// SIMATIC S7-200 SMART project (STEP 7-Micro/WIN SMART), CPU ST20

SYMBOL_TABLE Real_Sym
PressureDINT     VD100
PressureReal     VD104
PressRawMin      VD108
PressRawMax      VD112
PressFinalMin    VD116
PressFinalMax    VD120
PressureFinalVal VD124
TempDINT         VD128
TempReal         VD132
TempRawMin       VD136
TempRawMax       VD140
TempFinalMin     VD144
TempFinalMax     VD148
TempFinalVal     VD152
AutoPressureSV   VD156
AutoTempSV       VD160
NormPressSV      VD164
NormTempSV       VD168
RapidPressSV     VD172
RapidTempSV      VD176
OptPressSV       VD180
OptTempSV        VD184
TempErrorVal     VD188
TempErrorVal2    VD192
TempErrorValDINT VD196
HeaterOffTemp    VD200
PressureReal1    VD204
TempReal1        VD208
TempFinal1       VD212
PressureFinal1   VD216
VCCTolerance     VD220
VacuumLimit      VD224
VLTPressSV       VD228
TempRealPrint    VD232
TempDINTPrint    VD236
PressRealPrint   VD240
PressDINTPrint   VD244
END_SYMBOL_TABLE

SYMBOL_TABLE System Symbols
Always_On        SM0.0    // Always ON
Clock_1s         SM0.5    // Clock pulse that is ON for 0.5 s, OFF for 0.5 s, for a duty cycle time of 1 s.
END_SYMBOL_TABLE

SYMBOL_TABLE Bool_Sym
AutoSel          M0.0
ManualSel        M0.1
VacPumpManCmd    M0.2
HeaterManCmd     M0.3
AirVentManCmd    M0.4
PunchDownManCmd  M0.5
PunchUpManCmd    M0.6
VacPumpAutoCmd   M1.0
HeaterAutoCmd    M1.1
AirVentAutoCmd   M1.2
PunchDownAutoCmd M1.3
PunchUpAutoCmd   M1.4
AlarmCmd         M1.5
NormalSel        M2.0
RapidSel         M2.1
OptChoiceSel     M2.2
VLTSel           M2.3
AutoStart        M2.4
StartHeaterAuto  M2.5
PreTreat         M2.6
Vacuum1Done      M2.7
HeatingDone      M3.0
Vacuum2Done      M3.1
Sterilization    M3.2
Aeration         M3.3
VentOut          M3.4
CycleDone        M3.5
Vacuum3Done      M3.6
StartPunch       M3.7
PunchDone        M4.0
CycleDoneFinal   M4.1
StopOut          M4.2
OutVar           M4.3
StartHoldTime    M4.4
VLTPass          M4.5
VLTFail          M4.6
HoldTimeDone     M4.7
ResetCycleCount  M5.0
VLTStart         M5.1
VLTDone          M5.2
VLTVacuuming     M5.3
VLTHoldStart     M5.4
VLTTestPass      M5.5
VLTTestFail      M5.6
VLTDoneFinal     M5.7
MBUs_Done        M6.0
END_SYMBOL_TABLE

SYMBOL_TABLE Int_Sym
AutoSterTimeSV   VW0
AutoAerateTimeSV VW2
NormSterTimeSV   VW4
NormAerateTimeSV VW6
RapidSterTimeSV  VW8
RapidAerateTimeSV VW10
OptSterTimeSV    VW12
OptAerateTimeSV  VW14
SterTimePV       VW16
AerateTimePV     VW18
TempErrorValInt  VW20
TempBlinkOffVal  VW22
TempBlinkOffTime VW24
TempBlinkOnTime  VW26
AerateTimeSecPV  VW28
SterTimeSecPV    VW30
PunchSV          VW32
PunchPV          VW34
ClockVar1        VW36
OnCount          VW38
OffCount         VW40
VacuumHoldTimeSV VW42
VacuumHoldTimePV VW44
HoldTimePVSec    VW46
AutoStatus       VW48
CycleCount       VW50
OptHoldTimeSV    VW52
AutoHoldTimeSV   VW54
NormHoldTimeSV   VW56
RapidHoldTimeSV  VW58
TempIntPrint     VW60
PressIntPrint    VW62
YearRead         VW1774
MonthRead        VW1778
DateRead         VW1782
HourRead         VW1762
MinuteRead       VW1766
SecondsRead      VW1770
MinutesSet       VW1460
SecondsSet       VW1462
HourSet          VW1464
YearSet          VW1470
MonthSet         VW1474
DateSet          VW1490
END_SYMBOL_TABLE

ORGANIZATION_BLOCK MAIN:OB1
TITLE=Program Comments
BEGIN
Network 1
// Network Comment
LD     Always_On:SM0.0
ITD    EM0_Input0:AIW16, PressureDINT:VD100
AENO
DTR    PressureDINT:VD100, PressureReal1:VD204
AENO
MOVR   PressureReal1:VD204, PressureReal:VD104
AENO
/R     100.0, PressureReal:VD104
AENO
CALL   Lin_Trafo:SBR1, PressureReal:VD104, PressRawMin:VD108, PressRawMax:VD112, PressFinalMin:VD116, PressFinalMax:VD120, PressureFinal1:VD216
Network 2
// Network Comment
LD     Always_On:SM0.0
ITD    EM0_Input1:AIW18, TempDINT:VD128
AENO
DTR    TempDINT:VD128, TempReal1:VD208
AENO
MOVR   TempReal1:VD208, TempReal:VD132
AENO
/R     100.0, TempReal:VD132
AENO
CALL   Lin_Trafo:SBR1, TempReal:VD132, TempRawMin:VD136, TempRawMax:VD140, TempFinalMin:VD144, TempFinalMax:VD148, TempFinal1:VD212
Network 3
// (network saved uncompiled; FBD cells follow)
// row 0: c5 [INC_W ]  c8 [MOV_R ]
// row 1: c1 [AND Always_On:SM0.0 Clock_1s:SM0.5 ]  c2 --  c3 [P ]  c4 --  c5 [ EN:=power@row1, IN:=ClockVar1:VW36, ENO=>power, OUT=>ClockVar1:VW36]  c6 --  c7 --  c8 [ EN:=power@row1, IN:=TempFinal1:VD212, ENO=>V?0, OUT=>TempFinalVal:VD152]
// row 2: c1 [box]  c5 [box]  c8 [box]
Network 4
// (network saved uncompiled; FBD cells follow)
// row 0: c5 [MOV_R ]  c8 [MOV_W ]
// row 1: c1 [>=I ClockVar1:VW36 2 ]  c2 --  c3 [P ]  c4 --  c5 [ EN:=power@row1, IN:=PressureFinal1:VD216, ENO=>power, OUT=>PressureFinalVal:VD124]  c6 --  c7 --  c8 [ EN:=power@row1, IN:=0, ENO=>V?0, OUT=>ClockVar1:VW36]
// row 2: c1 [box]  c5 [box]  c8 [box]
Network 5
// Vacuum Pump
LD     Always_On:SM0.0
=      L60.0
LD     AutoSel:M0.0
=      L63.7
LD     ManualSel:M0.1
=      L63.6
LD     VacPumpManCmd:M0.2
=      L63.5
LD     VacPumpAutoCmd:M1.0
=      L63.4
LDN    Always_On:SM0.0
=      L63.3
LD     L60.0
CALL   Auto_Manual:SBR2, L63.7, L63.6, L63.5, L63.4, L63.3, CPU_Output0:Q0.0
Network 6
// Heater
LD     Always_On:SM0.0
=      L60.0
LD     AutoSel:M0.0
=      L63.7
LD     ManualSel:M0.1
=      L63.6
LD     HeaterManCmd:M0.3
=      L63.5
LD     HeaterAutoCmd:M1.1
=      L63.4
LDN    Always_On:SM0.0
=      L63.3
LD     L60.0
CALL   Auto_Manual:SBR2, L63.7, L63.6, L63.5, L63.4, L63.3, CPU_Output2:Q0.2
Network 7
// Air Vent
LD     Always_On:SM0.0
=      L60.0
LD     AutoSel:M0.0
=      L63.7
LD     ManualSel:M0.1
=      L63.6
LD     AirVentManCmd:M0.4
=      L63.5
LD     AirVentAutoCmd:M1.2
=      L63.4
LDN    Always_On:SM0.0
=      L63.3
LD     L60.0
CALL   Auto_Manual:SBR2, L63.7, L63.6, L63.5, L63.4, L63.3, CPU_Output4:Q0.4
Network 8
// ETO Punch Down
LD     Always_On:SM0.0
=      L60.0
LD     AutoSel:M0.0
=      L63.7
LD     ManualSel:M0.1
=      L63.6
LD     PunchDownManCmd:M0.5
=      L63.5
LD     PunchDownAutoCmd:M1.3
=      L63.4
LDN    Always_On:SM0.0
=      L63.3
LD     L60.0
CALL   Auto_Manual:SBR2, L63.7, L63.6, L63.5, L63.4, L63.3, CPU_Output3:Q0.3
Network 9
// ETO Punch Up
LD     Always_On:SM0.0
=      L60.0
LD     AutoSel:M0.0
=      L63.7
LD     ManualSel:M0.1
=      L63.6
LD     PunchUpManCmd:M0.6
=      L63.5
LD     PunchUpAutoCmd:M1.4
=      L63.4
LDN    Always_On:SM0.0
=      L63.3
LD     L60.0
CALL   Auto_Manual:SBR2, L63.7, L63.6, L63.5, L63.4, L63.3, CPU_Output6:Q0.6
Network 10
// Alarm Output
LD     AutoSel:M0.0
A      AlarmCmd:M1.5
=      CPU_Output5:Q0.5
Network 11
LD     NormalSel:M2.0
AN     AutoStart:M2.4
LD     NormalSel:M2.0
A      AutoStart:M2.4
OLD
EU
MOVR   NormPressSV:VD164, AutoPressureSV:VD156
AENO
MOVR   NormTempSV:VD168, AutoTempSV:VD160
AENO
MOVW   NormSterTimeSV:VW4, AutoSterTimeSV:VW0
AENO
MOVW   NormAerateTimeSV:VW6, AutoAerateTimeSV:VW2
AENO
MOVW   NormHoldTimeSV:VW56, AutoHoldTimeSV:VW54
Network 12
LD     RapidSel:M2.1
AN     AutoStart:M2.4
LD     RapidSel:M2.1
A      AutoStart:M2.4
OLD
EU
MOVR   RapidPressSV:VD172, AutoPressureSV:VD156
AENO
MOVR   RapidTempSV:VD176, AutoTempSV:VD160
AENO
MOVW   RapidSterTimeSV:VW8, AutoSterTimeSV:VW0
AENO
MOVW   RapidAerateTimeSV:VW10, AutoAerateTimeSV:VW2
AENO
MOVW   RapidHoldTimeSV:VW58, AutoHoldTimeSV:VW54
Network 13
LD     OptChoiceSel:M2.2
AN     AutoStart:M2.4
LD     OptChoiceSel:M2.2
A      AutoStart:M2.4
OLD
EU
MOVR   OptPressSV:VD180, AutoPressureSV:VD156
AENO
MOVR   OptTempSV:VD184, AutoTempSV:VD160
AENO
MOVW   OptSterTimeSV:VW12, AutoSterTimeSV:VW0
AENO
MOVW   OptAerateTimeSV:VW14, AutoAerateTimeSV:VW2
AENO
MOVW   OptHoldTimeSV:VW52, AutoHoldTimeSV:VW54
Network 14
LD     Always_On:SM0.0
CALL   AutoCycle:SBR0
Network 15
// (network saved uncompiled; FBD cells follow)
// row 0: c3 [MOV_W ]
// row 1: c1 [P ResetCycleCount:M5.0 ]  c2 --  c3 [ EN:=power@row1, IN:=0, ENO=>V?0, OUT=>CycleCount:VW50]
// row 2: c3 [box]
Network 16
LD     Always_On:SM0.0
CALL   VLT:SBR5
Network 17
LD     ManualSel:M0.1
EU
R      NormalSel:M2.0, 4
Network 18
LD     AutoSel:M0.0
A      VLTSel:M2.3
EU
R      NormalSel:M2.0, 3
Network 19
LD     AutoSel:M0.0
A      NormalSel:M2.0
EU
R      RapidSel:M2.1, 3
Network 20
LD     AutoSel:M0.0
A      RapidSel:M2.1
EU
R      NormalSel:M2.0, 1
R      OptChoiceSel:M2.2, 2
Network 21
LD     AutoSel:M0.0
A      OptChoiceSel:M2.2
EU
R      NormalSel:M2.0, 2
R      VLTSel:M2.3, 1
Network 22
// (network saved uncompiled; FBD cells follow)
// row 0: c1 [RTC ]
// row 1: c1 [ EN:=Always_On:SM0.0]
Network 23
// (network saved uncompiled; FBD cells follow)
// row 0: c1 [Print ]
// row 1: c1 [ EN:=Always_On:SM0.0]
END_ORGANIZATION_BLOCK

SUBROUTINE_BLOCK AutoCycle:SBR0
TITLE=Subroutine Comments
BEGIN
Network 1
// Network Comment
LD     AutoSel:M0.0
A      AutoStart:M2.4
EU
R      CPU_Output0:Q0.0, 7
Network 2
// Network Comment
// (network saved uncompiled; FBD cells follow)
// row 0: c5 [MOV_W ]  c8 [MOV_W ]  c11 [MOV_W ]  c14 [MOV_W ]  c17 [MOV_W ]
// row 1: c1 [AND AutoSel:M0.0 AutoStart:M2.4 ]  c2 --  c3 [P ]  c4 --  c5 [ EN:=power@row1, IN:=0, ENO=>power, OUT=>SterTimePV:VW16]  c6 --  c7 --  c8 [ EN:=power@row1, IN:=0, ENO=>power, OUT=>SterTimeSecPV:VW30]  c9 --  c10 --  c11 [ EN:=power@row1, IN:=0, ENO=>power, OUT=>HoldTimePVSec:VW46]  c12 --  c13 --  c14 [ EN:=power@row1, IN:=0, ENO=>power, OUT=>VacuumHoldTimePV:VW44]  c15 --  c16 --  c17 [ EN:=power@row1, IN:=0, ENO=>V?0, OUT=>PunchPV:VW34]
// row 2: c1 [box]  c5 [box]  c8 [box]  c11 [box]  c14 [box]  c17 [box]
Network 3
// Network Comment
LD     AutoSel:M0.0
A      AutoStart:M2.4
EU
MOVW   0, AerateTimePV:VW18
AENO
MOVW   0, AerateTimeSecPV:VW28
AENO
MOVW   0, AutoStatus:VW48
AENO
R      StartHeaterAuto:M2.5, 19
Network 4
LD     AutoSel:M0.0
A      AutoStart:M2.4
TON    T101, 10
Network 5
LD     AutoSel:M0.0
A      AutoStart:M2.4
A      T101
EU
MOVW   1, AutoStatus:VW48
AENO
S      PreTreat:M2.6, 1
Network 6
LD     AutoSel:M0.0
A      AutoStart:M2.4
A      T101
A      PreTreat:M2.6
EU
S      VacPumpAutoCmd:M1.0, 1
Network 7
LD     AutoSel:M0.0
A      AutoStart:M2.4
A      T101
A      VacPumpAutoCmd:M1.0
A      PreTreat:M2.6
TON    T102, 100
Network 8
// (network saved uncompiled; FBD cells follow)
// row 0: c1 [SUB_R ]
// row 1: c1 [ EN:=AutoStart:M2.4, IN1:=AutoTempSV:VD160, IN2:=-0.5, ENO=>V?0, OUT=>HeaterOffTemp:VD200]
// row 2: c1 [box]
// row 3: c1 [box]
Network 9
LDR<   TempFinalVal:VD152, AutoTempSV:VD160
A      AutoSel:M0.0
A      AutoStart:M2.4
A      T101
LD     T102
O      Vacuum1Done:M2.7
ALD
A      Always_On:SM0.0
EU
S      StartHeaterAuto:M2.5, 1
Network 10
LDR<=  PressureFinalVal:VD124, AutoPressureSV:VD156
A      AutoSel:M0.0
A      AutoStart:M2.4
A      VacPumpAutoCmd:M1.0
ON     AutoSel:M0.0
ON     AutoStart:M2.4
ON     PreTreat:M2.6
EU
R      VacPumpAutoCmd:M1.0, 1
Network 11
LDR<=  PressureFinalVal:VD124, AutoPressureSV:VD156
A      AutoSel:M0.0
A      AutoStart:M2.4
A      PreTreat:M2.6
EU
S      Vacuum1Done:M2.7, 1
Network 12
LDR>   TempFinalVal:VD152, HeaterOffTemp:VD200
A      StartHeaterAuto:M2.5
ON     AutoSel:M0.0
ON     AutoStart:M2.4
ON     Always_On:SM0.0
EU
R      StartHeaterAuto:M2.5, 1
Network 13
// (network saved uncompiled; FBD cells follow)
// row 0: c1 [SUB_R ]  c4 [MUL_R ]  c7 [ROUND ]  c10 [DI_I ]
// row 1: c1 [ EN:=StartHeaterAuto:M2.5, IN1:=AutoTempSV:VD160, IN2:=TempFinalVal:VD152, ENO=>power, OUT=>TempErrorVal:VD188]  c2 --  c3 --  c4 [ EN:=power@row1, IN1:=TempErrorVal:VD188, IN2:=0.5, ENO=>power, OUT=>TempErrorVal2:VD192]  c5 --  c6 --  c7 [ EN:=power@row1, IN:=TempErrorVal2:VD192, ENO=>power, OUT=>TempErrorValDINT:VD196]  c8 --  c9 --  c10 [ EN:=power@row1, IN:=TempErrorValDINT:VD196, ENO=>V?0, OUT=>TempErrorValInt:VW20]
// row 2: c1 [box]  c4 [box]  c7 [box]  c10 [box]
// row 3: c1 [box]  c4 [box]
Network 14
// (network saved uncompiled; FBD cells follow)
// row 0: c1 [SUB_I ]
// row 1: c1 [ EN:=StartHeaterAuto:M2.5, IN1:=+10, IN2:=TempErrorValInt:VW20, ENO=>V?0, OUT=>TempBlinkOffVal:VW22]
// row 2: c1 [box]
// row 3: c1 [box]
Network 15
// (network saved uncompiled; FBD cells follow)
// row 0: c3 [MOV_W ]
// row 1: c1 [<=I TempBlinkOffVal:VW22 2 ]  c2 --  c3 [ EN:=power@row1, IN:=2, ENO=>V?0, OUT=>TempBlinkOffTime:VW24]
// row 2: c1 [box]  c3 [box]
Network 16
// (network saved uncompiled; FBD cells follow)
// row 0: c3 [MOV_W ]
// row 1: c1 [>=I TempBlinkOffVal:VW22 8 ]  c2 --  c3 [ EN:=power@row1, IN:=8, ENO=>V?0, OUT=>TempBlinkOffTime:VW24]
// row 2: c1 [box]  c3 [box]
Network 17
// (network saved uncompiled; FBD cells follow)
// row 0: c4 [MOV_W ]
// row 1: c1 [>I TempBlinkOffVal:VW22 2 ]  c2 [AND ]  c3 --  c4 [ EN:=power@row1, IN:=TempBlinkOffVal:VW22, ENO=>V?0, OUT=>TempBlinkOffTime:VW24]
// row 2: c1 [box]  c2 [box]  c4 [box]
// row 3: c1 [<I TempBlinkOffVal:VW22 8 ]  c2 [box]
// row 4: c1 [box]
Network 18
// (network saved uncompiled; FBD cells follow)
// row 0: c3 [MOV_W ]
// row 1: c1 [<I TempErrorValInt:VW20 5 ]  c2 --  c3 [ EN:=power@row1, IN:=5, ENO=>V?0, OUT=>TempBlinkOnTime:VW26]
// row 2: c1 [box]  c3 [box]
Network 19
// (network saved uncompiled; FBD cells follow)
// row 0: c3 [MOV_W ]
// row 1: c1 [>I TempErrorValInt:VW20 7 ]  c2 --  c3 [ EN:=power@row1, IN:=8, ENO=>V?0, OUT=>TempBlinkOnTime:VW26]
// row 2: c1 [box]  c3 [box]
Network 20
// (network saved uncompiled; FBD cells follow)
// row 0: c4 [MOV_W ]
// row 1: c1 [>=I TempErrorValInt:VW20 5 ]  c2 [AND ]  c3 --  c4 [ EN:=power@row1, IN:=TempErrorValInt:VW20, ENO=>V?0, OUT=>TempBlinkOnTime:VW26]
// row 2: c1 [box]  c2 [box]  c4 [box]
// row 3: c1 [<=I TempErrorValInt:VW20 7 ]  c2 [box]
// row 4: c1 [box]
Network 21
LD     Always_On:SM0.0
A      PreTreat:M2.6
CALL   BlinkSBR:SBR4
Network 22
LDR>=  TempFinalVal:VD152, AutoTempSV:VD160
A      AutoSel:M0.0
A      AutoStart:M2.4
A      PreTreat:M2.6
A      Vacuum1Done:M2.7
AN     VLTFail:M4.6
AN     CycleDone:M3.5
EU
S      HeatingDone:M3.0, 1
S      StartHoldTime:M4.4, 1
Network 23
// (network saved uncompiled; FBD cells follow)
// row 0: c5 [MOV_W ]
// row 1: c1 [AND AutoSel:M0.0 AutoStart:M2.4 Vacuum1Done:M2.7 HeatingDone:M3.0 StartHoldTime:M4.4 VLTFail:M4.6 CycleDone:M3.5 ]  c2 --  c3 [P ]  c4 --  c5 [ EN:=power@row1, IN:=2, ENO=>V?0, OUT=>AutoStatus:VW48]
// row 2: c1 [box]  c5 [box]
// row 3: c1 [box]
// row 4: c1 [box]
// row 5: c1 [box]
// row 6: c1 [box]
// row 7: c1 [box]
Network 24
// (network saved uncompiled; FBD cells follow)
// row 0: c5 [INC_W ]
// row 1: c1 [AND StartHoldTime:M4.4 AutoSel:M0.0 AutoStart:M2.4 Vacuum1Done:M2.7 HeatingDone:M3.0 Clock_1s:SM0.5 ]  c2 --  c3 [P ]  c4 --  c5 [ EN:=power@row1, IN:=HoldTimePVSec:VW46, ENO=>V?0, OUT=>HoldTimePVSec:VW46]
// row 2: c1 [box]  c5 [box]
// row 3: c1 [box]
// row 4: c1 [box]
// row 5: c1 [box]
// row 6: c1 [box]
Network 25
// (network saved uncompiled; FBD cells follow)
// row 0: c6 [INC_W ]  c9 [MOV_W ]
// row 1: c1 [>=I HoldTimePVSec:VW46 60 ]  c2 [AND StartHoldTime:M4.4 AutoStart:M2.4 ]  c3 --  c4 [P ]  c5 --  c6 [ EN:=power@row1, IN:=VacuumHoldTimePV:VW44, ENO=>power, OUT=>VacuumHoldTimePV:VW44]  c7 --  c8 --  c9 [ EN:=power@row1, IN:=0, ENO=>V?0, OUT=>HoldTimePVSec:VW46]
// row 2: c1 [box]  c2 [box]  c6 [box]  c9 [box]
// row 3: c2 [box]
// row 4: c2 [box]
Network 26
LDW>=  VacuumHoldTimePV:VW44, AutoHoldTimeSV:VW54
A      StartHoldTime:M4.4
AN     CycleDone:M3.5
EU
S      HoldTimeDone:M4.7, 1
Network 27
// (network saved uncompiled; FBD cells follow)
// row 0: c1 [ADD_R ]
// row 1: c1 [ EN:=AutoStart:M2.4, IN1:=AutoPressureSV:VD156, IN2:=VCCTolerance:VD220, ENO=>V?0, OUT=>VacuumLimit:VD224]
// row 2: c1 [box]
// row 3: c1 [box]
Network 28
LDR>   PressureFinalVal:VD124, VacuumLimit:VD224
A      Vacuum1Done:M2.7
A      HeatingDone:M3.0
A      PreTreat:M2.6
A      StartHoldTime:M4.4
AN     HoldTimeDone:M4.7
EU
S      VLTFail:M4.6, 1
R      VLTPass:M4.5, 1
Network 29
LDR<=  PressureFinalVal:VD124, VacuumLimit:VD224
A      AutoStart:M2.4
A      StartHoldTime:M4.4
A      HoldTimeDone:M4.7
A      HeatingDone:M3.0
A      Vacuum1Done:M2.7
AN     VLTFail:M4.6
AN     CycleDone:M3.5
EU
S      VLTPass:M4.5, 1
Network 30
LD     AutoStart:M2.4
A      Vacuum1Done:M2.7
A      HeatingDone:M3.0
A      PreTreat:M2.6
A      StartHoldTime:M4.4
A      HoldTimeDone:M4.7
A      VLTPass:M4.5
AN     VLTFail:M4.6
AN     CycleDone:M3.5
EU
S      Vacuum2Done:M3.1, 1
R      StartHoldTime:M4.4, 1
Network 31
LD     Vacuum1Done:M2.7
A      HeatingDone:M3.0
A      PreTreat:M2.6
A      AutoSel:M0.0
A      AutoStart:M2.4
A      Vacuum2Done:M3.1
AN     CycleDone:M3.5
EU
MOVW   3, AutoStatus:VW48
AENO
R      PreTreat:M2.6, 1
S      StartPunch:M3.7, 1
Network 32
LD     StartPunch:M3.7
A      AutoStart:M2.4
EU
S      PunchDownAutoCmd:M1.3, 1
Network 33
// (network saved uncompiled; FBD cells follow)
// row 0: c5 [INC_W ]
// row 1: c1 [AND PunchDownAutoCmd:M1.3 StartPunch:M3.7 ]  c2 --  c3 [P ]  c4 --  c5 [ EN:=power@row1, IN:=PunchPV:VW34, ENO=>V?0, OUT=>PunchPV:VW34]
// row 2: c1 [box]  c5 [box]
Network 34
LD     PunchDownAutoCmd:M1.3
A      StartPunch:M3.7
TON    T103, 20
Network 35
LD     PunchDownAutoCmd:M1.3
A      StartPunch:M3.7
A      T103
EU
R      PunchDownAutoCmd:M1.3, 1
S      PunchUpAutoCmd:M1.4, 1
Network 36
LD     PunchUpAutoCmd:M1.4
A      StartPunch:M3.7
TON    T104, 10
Network 37
LDW<   PunchPV:VW34, PunchSV:VW32
A      StartPunch:M3.7
A      T104
A      PunchUpAutoCmd:M1.4
EU
S      PunchDownAutoCmd:M1.3, 1
Network 38
LD     PunchUpAutoCmd:M1.4
A      StartPunch:M3.7
A      T104
EU
R      PunchUpAutoCmd:M1.4, 1
Network 39
LDW>=  PunchPV:VW34, PunchSV:VW32
A      StartPunch:M3.7
AN     PunchDownAutoCmd:M1.3
AN     PunchUpAutoCmd:M1.4
TON    T105, 10
Network 40
LDW>=  PunchPV:VW34, PunchSV:VW32
A      StartPunch:M3.7
AN     PunchDownAutoCmd:M1.3
AN     PunchUpAutoCmd:M1.4
A      T105
A      VLTPass:M4.5
AN     CycleDone:M3.5
EU
R      StartPunch:M3.7, 1
S      Sterilization:M3.2, 1
S      PunchDone:M4.0, 1
Network 41
// (network saved uncompiled; FBD cells follow)
// row 0: c5 [MOV_W ]  c8 [MOV_W ]
// row 1: c1 [AND Sterilization:M3.2 AutoStart:M2.4 VLTFail:M4.6 ]  c2 --  c3 [P ]  c4 --  c5 [ EN:=power@row1, IN:=0, ENO=>power, OUT=>SterTimePV:VW16]  c6 --  c7 --  c8 [ EN:=power@row1, IN:=4, ENO=>V?0, OUT=>AutoStatus:VW48]
// row 2: c1 [box]  c5 [box]  c8 [box]
// row 3: c1 [box]
Network 42
// (network saved uncompiled; FBD cells follow)
// row 0: c5 [INC_W ]
// row 1: c1 [AND Sterilization:M3.2 Clock_1s:SM0.5 ]  c2 --  c3 [P ]  c4 --  c5 [ EN:=power@row1, IN:=SterTimeSecPV:VW30, ENO=>V?0, OUT=>SterTimeSecPV:VW30]
// row 2: c1 [box]  c5 [box]
Network 43
// (network saved uncompiled; FBD cells follow)
// row 0: c6 [INC_W ]  c9 [MOV_W ]
// row 1: c1 [>=I SterTimeSecPV:VW30 60 ]  c2 [AND Sterilization:M3.2 ]  c3 --  c4 [P ]  c5 --  c6 [ EN:=power@row1, IN:=SterTimePV:VW16, ENO=>power, OUT=>SterTimePV:VW16]  c7 --  c8 --  c9 [ EN:=power@row1, IN:=0, ENO=>V?0, OUT=>SterTimeSecPV:VW30]
// row 2: c1 [box]  c2 [box]  c6 [box]  c9 [box]
// row 3: c2 [box]
Network 44
LDW>=  SterTimePV:VW16, AutoSterTimeSV:VW0
A      Sterilization:M3.2
A      AutoStart:M2.4
A      AutoSel:M0.0
A      Vacuum1Done:M2.7
A      HeatingDone:M3.0
A      Vacuum2Done:M3.1
A      VLTPass:M4.5
AN     CycleDone:M3.5
EU
MOVW   5, AutoStatus:VW48
AENO
R      Sterilization:M3.2, 1
S      Aeration:M3.3, 1
Network 45
LDR>   PressureFinalVal:VD124, AutoPressureSV:VD156
A      Aeration:M3.3
A      AutoStart:M2.4
AN     CycleDone:M3.5
EU
S      VacPumpAutoCmd:M1.0, 1
Network 46
LDR<=  PressureFinalVal:VD124, AutoPressureSV:VD156
A      Aeration:M3.3
A      VacPumpAutoCmd:M1.0
A      AutoStart:M2.4
EU
R      VacPumpAutoCmd:M1.0, 1
S      Vacuum3Done:M3.6, 1
Network 47
// (network saved uncompiled; FBD cells follow)
// row 0: c5 [INC_W ]
// row 1: c1 [AND Aeration:M3.3 Clock_1s:SM0.5 ]  c2 --  c3 [P ]  c4 --  c5 [ EN:=power@row1, IN:=AerateTimeSecPV:VW28, ENO=>V?0, OUT=>AerateTimeSecPV:VW28]
// row 2: c1 [box]  c5 [box]
Network 48
// Increase Aeration Time after every minute
// (network saved uncompiled; FBD cells follow)
// row 0: c6 [INC_W ]  c9 [MOV_W ]
// row 1: c1 [>=I AerateTimeSecPV:VW28 60 ]  c2 [AND Aeration:M3.3 ]  c3 --  c4 [P ]  c5 --  c6 [ EN:=power@row1, IN:=AerateTimePV:VW18, ENO=>power, OUT=>AerateTimePV:VW18]  c7 --  c8 --  c9 [ EN:=power@row1, IN:=0, ENO=>V?0, OUT=>AerateTimeSecPV:VW28]
// row 2: c1 [box]  c2 [box]  c6 [box]  c9 [box]
// row 3: c2 [box]
Network 49
// If aeration time is completed then reset Aeration bit, it will reset Vacuum command if it is still running
LDW>=  AerateTimePV:VW18, AutoAerateTimeSV:VW2
A      Aeration:M3.3
EU
R      Aeration:M3.3, 1
Network 50
LDN    Aeration:M3.3
A      Vacuum3Done:M3.6
LD     VLTFail:M4.6
A      AutoStart:M2.4
OLD
ON     Always_On:SM0.0
A      Vacuum1Done:M2.7
A      HeatingDone:M3.0
EU
S      VentOut:M3.4, 1
Network 51
// (network saved uncompiled; FBD cells follow)
// row 0: c5 [MOV_W ]
// row 1: c1 [AND VentOut:M3.4 VLTFail:M4.6 ]  c2 --  c3 [P ]  c4 --  c5 [ EN:=power@row1, IN:=6, ENO=>V?0, OUT=>AutoStatus:VW48]
// row 2: c1 [box]  c5 [box]
Network 52
LD     VentOut:M3.4
A      AutoStart:M2.4
A      AutoStart:M2.4
A      Vacuum1Done:M2.7
A      HeatingDone:M3.0
EU
S      AirVentAutoCmd:M1.2, 1
Network 53
// Set CycleDone and Alarm when Pressure reaches above -50 to alert the operator, Air Vent is still on
LDR>=  PressureFinalVal:VD124, -10.0
A      VentOut:M3.4
A      AirVentAutoCmd:M1.2
A      AutoStart:M2.4
A      Vacuum1Done:M2.7
A      HeatingDone:M3.0
EU
S      CycleDone:M3.5, 1
Network 54
LD     CycleDone:M3.5
A      AutoStart:M2.4
EU
S      AlarmCmd:M1.5, 1
Network 55
// (network saved uncompiled; FBD cells follow)
// row 0: c5 [MOV_W ]  c8 [INC_W ]
// row 1: c1 [AND CycleDone:M3.5 AutoStart:M2.4 VLTFail:M4.6 Vacuum1Done:M2.7 HeatingDone:M3.0 ]  c2 --  c3 [P ]  c4 --  c5 [ EN:=power@row1, IN:=7, ENO=>power, OUT=>AutoStatus:VW48]  c6 --  c7 --  c8 [ EN:=power@row1, IN:=CycleCount:VW50, ENO=>V?0, OUT=>CycleCount:VW50]
// row 2: c1 [box]  c5 [box]  c8 [box]
// row 3: c1 [box]
// row 4: c1 [box]
// row 5: c1 [box]
Network 56
// (network saved uncompiled; FBD cells follow)
// row 0: c3 [MOV_W ]
// row 1: c1 [P VLTFail:M4.6 ]  c2 --  c3 [ EN:=power@row1, IN:=8, ENO=>V?0, OUT=>AutoStatus:VW48]
// row 2: c3 [box]
Network 57
// reset VentOut and CycleDone when Pressure reaches more than -5 (almost zero)
LDR>=  PressureFinalVal:VD124, -5.0
A      VentOut:M3.4
A      AirVentAutoCmd:M1.2
EU
R      VentOut:M3.4, 2
S      CycleDoneFinal:M4.1, 1
R      AirVentAutoCmd:M1.2, 1
Network 58
// When Cycle finally done, reset all done bits and also reset alarm
LD     CycleDoneFinal:M4.1
A      AutoStart:M2.4
R      AutoStart:M2.4, 13
R      AlarmCmd:M1.5, 1
Network 59
// reset all bits from autostart till cycleDoneFinal
LDN    AutoSel:M0.0
ON     AutoStart:M2.4
R      AutoStart:M2.4, 19
Network 60
// Reset Sterilization and Aeration times
// (network saved uncompiled; FBD cells follow)
// row 0: c5 [MOV_W ]  c8 [MOV_W ]  c11 [MOV_W ]  c14 [MOV_W ]
// row 1: c1 [OR AutoSel:M0.0 AutoStart:M2.4 ]  c2 --  c3 [P ]  c4 --  c5 [ EN:=power@row1, IN:=0, ENO=>power, OUT=>SterTimePV:VW16]  c6 --  c7 --  c8 [ EN:=power@row1, IN:=0, ENO=>power, OUT=>AerateTimePV:VW18]  c9 --  c10 --  c11 [ EN:=power@row1, IN:=0, ENO=>power, OUT=>PunchPV:VW34]  c12 --  c13 --  c14 [ EN:=power@row1, IN:=0, ENO=>V?0, OUT=>VacuumHoldTimePV:VW44]
// row 2: c1 [box]  c5 [box]  c8 [box]  c11 [box]  c14 [box]
Network 61
LDN    AutoSel:M0.0
ON     AutoStart:M2.4
EU
R      CPU_Output0:Q0.0, 7
Network 62
LDN    AutoSel:M0.0
ON     AutoStart:M2.4
EU
R      VacPumpAutoCmd:M1.0, 6
END_SUBROUTINE_BLOCK

// SBR1: protected block, not included

// SBR2: protected block, not included

// SBR3: protected block, not included

SUBROUTINE_BLOCK BlinkSBR:SBR4
TITLE=Subroutine Comments
BEGIN
Network 1
// Network Comment
LD     Always_On:SM0.0
A      StartHeaterAuto:M2.5
EU
S      OutVar:M4.3, 1
Network 2
// (network saved uncompiled; FBD cells follow)
// row 0: c5 [INC_W ]
// row 1: c1 [AND StartHeaterAuto:M2.5 Clock_1s:SM0.5 OutVar:M4.3 ]  c2 --  c3 [P ]  c4 --  c5 [ EN:=power@row1, IN:=OnCount:VW38, ENO=>V?0, OUT=>OnCount:VW38]
// row 2: c1 [box]  c5 [box]
// row 3: c1 [box]
Network 3
LDW>=  OnCount:VW38, TempBlinkOnTime:VW26
EU
R      OutVar:M4.3, 1
Network 4
LDW>=  OnCount:VW38, TempBlinkOnTime:VW26
S      StopOut:M4.2, 1
Network 5
// (network saved uncompiled; FBD cells follow)
// row 0: c3 [MOV_W ]
// row 1: c1 [>=I OnCount:VW38 TempBlinkOnTime:VW26 ]  c2 --  c3 [ EN:=power@row1, IN:=0, ENO=>V?0, OUT=>OnCount:VW38]
// row 2: c1 [box]  c3 [box]
Network 6
// (network saved uncompiled; FBD cells follow)
// row 0: c5 [INC_W ]
// row 1: c1 [AND StartHeaterAuto:M2.5 Clock_1s:SM0.5 StopOut:M4.2 ]  c2 --  c3 [P ]  c4 --  c5 [ EN:=power@row1, IN:=OffCount:VW40, ENO=>V?0, OUT=>OffCount:VW40]
// row 2: c1 [box]  c5 [box]
// row 3: c1 [box]
Network 7
LDW>=  OffCount:VW40, TempBlinkOffTime:VW24
EU
R      StopOut:M4.2, 1
Network 8
LDW>=  OffCount:VW40, TempBlinkOffTime:VW24
EU
S      OutVar:M4.3, 1
Network 9
// (network saved uncompiled; FBD cells follow)
// row 0: c3 [MOV_W ]
// row 1: c1 [>=I OffCount:VW40 TempBlinkOffTime:VW24 ]  c2 --  c3 [ EN:=power@row1, IN:=0, ENO=>V?0, OUT=>OffCount:VW40]
// row 2: c1 [box]  c3 [box]
Network 10
LDR>   TempFinalVal:VD152, HeaterOffTemp:VD200
AN     StartHeaterAuto:M2.5
R      OutVar:M4.3, 1
Network 11
// (network saved uncompiled; FBD cells follow)
// row 0: c1 [MOV_W ]  c4 [MOV_W ]
// row 1: c1 [EN StartHeaterAuto:M2.5 IN:=0, ENO=>power, OUT=>OffCount:VW40]  c2 --  c3 --  c4 [ EN:=power@row1, IN:=0, ENO=>V?0, OUT=>OnCount:VW38]
// row 2: c1 [box]  c4 [box]
Network 12
LD     StartHeaterAuto:M2.5
A      OutVar:M4.3
=      HeaterAutoCmd:M1.1
Network 17
// Network Comment
END_SUBROUTINE_BLOCK

SUBROUTINE_BLOCK VLT:SBR5
TITLE=Subroutine Comments
BEGIN
Network 1
LD     AutoSel:M0.0
A      VLTStart:M5.1
A      VLTSel:M2.3
EU
MOVW   0, VacuumHoldTimePV:VW44
AENO
MOVW   0, HoldTimePVSec:VW46
AENO
R      CPU_Output0:Q0.0, 7
R      VLTDone:M5.2, 6
Network 2
LDR>=  PressureFinalVal:VD124, VLTPressSV:VD228
A      VLTSel:M2.3
A      VLTStart:M5.1
A      AutoSel:M0.0
AN     VLTHoldStart:M5.4
AN     VLTDone:M5.2
AN     VLTTestFail:M5.6
AN     VLTTestPass:M5.5
EU
S      VacPumpAutoCmd:M1.0, 1
S      VLTVacuuming:M5.3, 1
Network 3
LDR<   PressureFinalVal:VD124, VLTPressSV:VD228
A      VLTSel:M2.3
A      VLTStart:M5.1
A      AutoSel:M0.0
A      VacPumpAutoCmd:M1.0
EU
S      VLTHoldStart:M5.4, 1
R      VacPumpAutoCmd:M1.0, 1
R      VLTVacuuming:M5.3, 1
Network 4
// (network saved uncompiled; FBD cells follow)
// row 0: c5 [INC_W ]
// row 1: c1 [AND VLTSel:M2.3 VLTStart:M5.1 AutoSel:M0.0 VLTHoldStart:M5.4 Clock_1s:SM0.5 ]  c2 --  c3 [P ]  c4 --  c5 [ EN:=power@row1, IN:=HoldTimePVSec:VW46, ENO=>V?0, OUT=>HoldTimePVSec:VW46]
// row 2: c1 [box]  c5 [box]
// row 3: c1 [box]
// row 4: c1 [box]
// row 5: c1 [box]
Network 5
// (network saved uncompiled; FBD cells follow)
// row 0: c6 [INC_W ]  c9 [MOV_W ]
// row 1: c1 [>=I HoldTimePVSec:VW46 60 ]  c2 [AND VLTHoldStart:M5.4 VLTStart:M5.1 AutoSel:M0.0 VLTSel:M2.3 ]  c3 --  c4 [P ]  c5 --  c6 [ EN:=power@row1, IN:=VacuumHoldTimePV:VW44, ENO=>power, OUT=>VacuumHoldTimePV:VW44]  c7 --  c8 --  c9 [ EN:=power@row1, IN:=0, ENO=>V?0, OUT=>HoldTimePVSec:VW46]
// row 2: c1 [box]  c2 [box]  c6 [box]  c9 [box]
// row 3: c2 [box]
// row 4: c2 [box]
// row 5: c2 [box]
// row 6: c2 [box]
Network 6
LDW>=  VacuumHoldTimePV:VW44, VacuumHoldTimeSV:VW42
A      VLTHoldStart:M5.4
A      VLTStart:M5.1
A      AutoSel:M0.0
LD     VLTSel:M2.3
A      VLTTestFail:M5.6
OLD
EU
S      VLTDone:M5.2, 1
Network 7
// (network saved uncompiled; FBD cells follow)
// row 0: c1 [ADD_R ]
// row 1: c1 [ EN:=VLTStart:M5.1, IN1:=VLTPressSV:VD228, IN2:=VCCTolerance:VD220, ENO=>V?0, OUT=>VacuumLimit:VD224]
// row 2: c1 [box]
// row 3: c1 [box]
Network 8
LDR>   PressureFinalVal:VD124, VacuumLimit:VD224
A      VLTHoldStart:M5.4
A      VLTSel:M2.3
A      VLTStart:M5.1
A      AutoSel:M0.0
AN     VLTDone:M5.2
EU
S      VLTTestFail:M5.6, 1
R      VLTTestPass:M5.5, 1
R      VLTHoldStart:M5.4, 1
Network 9
LDR<=  PressureFinalVal:VD124, VacuumLimit:VD224
A      VLTStart:M5.1
A      VLTHoldStart:M5.4
A      VLTDone:M5.2
AN     VLTTestFail:M5.6
A      AutoSel:M0.0
A      VLTSel:M2.3
EU
S      VLTTestPass:M5.5, 1
R      VLTHoldStart:M5.4, 1
Network 10
// after VLTDone and Pass/Fail determination, vent out, reset VLTStart and all other variables and outputs
LD     VLTDone:M5.2
A      VLTStart:M5.1
A      VLTSel:M2.3
A      AutoSel:M0.0
EU
S      AirVentAutoCmd:M1.2, 1
Network 11
LDR>=  PressureFinalVal:VD124, -10.0
A      VLTStart:M5.1
A      AirVentAutoCmd:M1.2
EU
S      VLTDoneFinal:M5.7, 1
R      AirVentAutoCmd:M1.2, 1
Network 12
LD     VLTDoneFinal:M5.7
A      VLTSel:M2.3
A      VLTStart:M5.1
EU
MOVW   0, VacuumHoldTimePV:VW44
AENO
R      VLTStart:M5.1, 7
R      CPU_Output0:Q0.0, 7
Network 13
LDN    AutoSel:M0.0
ON     VLTStart:M5.1
EU
R      VacPumpAutoCmd:M1.0, 6
R      VLTDone:M5.2, 1
END_SUBROUTINE_BLOCK

// SBR6: protected block, not included

SUBROUTINE_BLOCK RTC:SBR7
TITLE=SUBROUTINE COMMENTS
BEGIN
Network 1
// Network Title
// Network Comment
LD     T249
R      M8.0, 1
Network 2
LD     M8.0
TON    T249, +100
Network 3
// (network saved uncompiled; FBD cells follow)
// row 0: c3 [SET_RTC ]
// row 1: c1 [OR M8.0 M9.0 ]  c2 --  c3 [ EN:=power@row1, T:=VB800, ENO=>V?0]
// row 2: c1 [box]  c3 [box]
Network 4
// (network saved uncompiled; FBD cells follow)
// row 0: c3 [READ_RTC ]
// row 1: c1 [AND Always_On:SM0.0 M8.0 M9.0 ]  c2 --  c3 [ EN:=power@row1, T:=VB800, ENO=>V?0]
// row 2: c1 [box]  c3 [box]
// row 3: c1 [box]
Network 5
// (network saved uncompiled; FBD cells follow)
// row 0: c4 [B_I ]  c7 [BCD_I ]
// row 1: c1 [AND Always_On:SM0.0 M8.0 ]  c2 -- v  c3 --  c4 [ EN:=power@row1, IN:=VB803, ENO=>power, OUT=>VW1760]  c5 --  c6 --  c7 [ EN:=power@row1, IN:=VW1760, ENO=>V?0, OUT=>HourRead:VW1762]
// row 2: c1 [box]  c2 ^v  c4 [box]  c7 [box]
// row 3: c2 ^v  c4 [B_I ]  c7 [BCD_I ]
// row 4: c2 ^v  c3 --  c4 [ EN:=power@row4, IN:=VB804, ENO=>power, OUT=>VW1764]  c5 --  c6 --  c7 [ EN:=power@row4, IN:=VW1764, ENO=>V?0, OUT=>MinuteRead:VW1766]
// row 5: c2 ^v  c4 [box]  c7 [box]
// row 6: c2 ^v  c4 [B_I ]  c7 [BCD_I ]
// row 7: c2 ^  c3 --  c4 [ EN:=power@row7, IN:=VB805, ENO=>power, OUT=>VW1768]  c5 --  c6 --  c7 [ EN:=power@row7, IN:=VW1768, ENO=>V?0, OUT=>SecondsRead:VW1770]
// row 8: c4 [box]  c7 [box]
Network 6
// (network saved uncompiled; FBD cells follow)
// row 0: c4 [B_I ]  c7 [BCD_I ]
// row 1: c1 [AND Always_On:SM0.0 M9.0 ]  c2 -- v  c3 --  c4 [ EN:=power@row1, IN:=VB800, ENO=>power, OUT=>VW1772]  c5 --  c6 --  c7 [ EN:=power@row1, IN:=VW1772, ENO=>V?0, OUT=>YearRead:VW1774]
// row 2: c1 [box]  c2 ^v  c4 [box]  c7 [box]
// row 3: c2 ^v  c4 [B_I ]  c7 [BCD_I ]
// row 4: c2 ^v  c3 --  c4 [ EN:=power@row4, IN:=VB801, ENO=>power, OUT=>VW1776]  c5 --  c6 --  c7 [ EN:=power@row4, IN:=VW1776, ENO=>V?0, OUT=>MonthRead:VW1778]
// row 5: c2 ^v  c4 [box]  c7 [box]
// row 6: c2 ^v  c4 [B_I ]  c7 [BCD_I ]
// row 7: c2 ^  c3 --  c4 [ EN:=power@row7, IN:=VB802, ENO=>power, OUT=>VW1780]  c5 --  c6 --  c7 [ EN:=power@row7, IN:=VW1780, ENO=>V?0, OUT=>DateRead:VW1782]
// row 8: c4 [box]  c7 [box]
Network 7
// (network saved uncompiled; FBD cells follow)
// row 0: c4 [I_BCD ]  c7 [I_B ]
// row 1: c1 [AND M8.0 ]  c2 -- v  c3 --  c4 [ EN:=power@row1, IN:=MinutesSet:VW1460, ENO=>power, OUT=>VW1452]  c5 --  c6 --  c7 [ EN:=power@row1, IN:=VW1452, ENO=>V?0, OUT=>VB804]
// row 2: c2 ^v  c4 [box]  c7 [box]
// row 3: c2 ^v  c4 [I_BCD ]  c7 [I_B ]
// row 4: c2 ^v  c3 --  c4 [ EN:=power@row4, IN:=HourSet:VW1464, ENO=>power, OUT=>VW1450]  c5 --  c6 --  c7 [ EN:=power@row4, IN:=VW1450, ENO=>V?0, OUT=>VB803]
// row 5: c2 ^v  c4 [box]  c7 [box]
// row 6: c2 ^v  c4 [I_BCD ]  c7 [I_B ]
// row 7: c2 ^  c3 --  c4 [ EN:=power@row7, IN:=SecondsSet:VW1462, ENO=>power, OUT=>VW1454]  c5 --  c6 --  c7 [ EN:=power@row7, IN:=VW1454, ENO=>V?0, OUT=>VB805]
// row 8: c4 [box]  c7 [box]
Network 8
// (network saved uncompiled; FBD cells follow)
// row 0: c4 [I_BCD ]  c7 [I_B ]
// row 1: c1 [AND M9.0 ]  c2 -- v  c3 --  c4 [ EN:=power@row1, IN:=DateSet:VW1490, ENO=>power, OUT=>VW1468]  c5 --  c6 --  c7 [ EN:=power@row1, IN:=VW1468, ENO=>V?0, OUT=>VB802]
// row 2: c2 ^v  c4 [box]  c7 [box]
// row 3: c2 ^v  c4 [I_BCD ]  c7 [I_B ]
// row 4: c2 ^v  c3 --  c4 [ EN:=power@row4, IN:=YearSet:VW1470, ENO=>power, OUT=>VW1472]  c5 --  c6 --  c7 [ EN:=power@row4, IN:=VW1472, ENO=>V?0, OUT=>VB800]
// row 5: c2 ^v  c4 [box]  c7 [box]
// row 6: c2 ^v  c4 [I_BCD ]  c7 [I_B ]
// row 7: c2 ^  c3 --  c4 [ EN:=power@row7, IN:=MonthSet:VW1474, ENO=>power, OUT=>VW1476]  c5 --  c6 --  c7 [ EN:=power@row7, IN:=VW1476, ENO=>V?0, OUT=>VB801]
// row 8: c4 [box]  c7 [box]
Network 9
LD     M9.0
TON    T248, +100
Network 10
LD     T248
R      M9.0, 1
Network 25
// Network Comment
END_SUBROUTINE_BLOCK

SUBROUTINE_BLOCK Print:SBR8
TITLE=Subroutine Comments
BEGIN
Network 1
LD     Always_On:SM0.0
=      L60.0
LD     Always_On:SM0.0
=      L63.7
LD     L60.0
CALL   MBUS_SERVER:SBR6, L63.7, 502, 0, 0, 20, &VB400, MBUs_Done:M6.0, MB10
Network 2
// Network Comment
// (network saved uncompiled; FBD cells follow)
// row 0: c2 [MOV_W ]
// row 1: c1 [OR AutoStart:M2.4 VLTStart:M5.1 ]  c2 [ EN:=power@row1, IN:=1, ENO=>?0_20_0, OUT=>VW400]
// row 2: c1 [box]  c2 [box]
// row 3: c2 [box]
Network 3
// Network Comment
// (network saved uncompiled; FBD cells follow)
// row 0: c3 [MOV_W ]
// row 1: c1 [OR AutoStart:M2.4 VLTStart:M5.1 ]  c2 --  c3 [EN IN:=0, ENO=>V?0, OUT=>VW400]
// row 2: c1 [box]  c3 [box]
Network 4
// (network saved uncompiled; FBD cells follow)
// row 0: c1 [MOV_W ]
// row 1: c1 [ EN:=Always_On:SM0.0, IN:=DateRead:VW1782, ENO=>?0_20_0, OUT=>VW402]
// row 2: c1 [box]
Network 5
// (network saved uncompiled; FBD cells follow)
// row 0: c1 [MOV_W ]
// row 1: c1 [ EN:=Always_On:SM0.0, IN:=MonthRead:VW1778, ENO=>V?0, OUT=>VW404]
// row 2: c1 [box]
Network 6
// (network saved uncompiled; FBD cells follow)
// row 0: c1 [MOV_W ]
// row 1: c1 [ EN:=Always_On:SM0.0, IN:=YearRead:VW1774, ENO=>V?0, OUT=>VW406]
// row 2: c1 [box]
Network 7
// (network saved uncompiled; FBD cells follow)
// row 0: c1 [MOV_W ]
// row 1: c1 [ EN:=Always_On:SM0.0, IN:=HourRead:VW1762, ENO=>V?0, OUT=>VW408]
// row 2: c1 [box]
Network 8
// (network saved uncompiled; FBD cells follow)
// row 0: c1 [MOV_W ]
// row 1: c1 [ EN:=Always_On:SM0.0, IN:=MinuteRead:VW1766, ENO=>V?0, OUT=>VW410]
// row 2: c1 [box]
Network 9
// (network saved uncompiled; FBD cells follow)
// row 0: c1 [MUL_R ]  c3 [ROUND ]  c5 [DI_I ]  c7 [MOV_W ]
// row 1: c1 [ EN:=Always_On:SM0.0, IN1:=TempFinalVal:VD152, IN2:=10.0, ENO=>power, OUT=>TempRealPrint:VD232]  c2 --  c3 [ EN:=power@row1, IN:=TempRealPrint:VD232, ENO=>power, OUT=>TempDINTPrint:VD236]  c4 --  c5 [ EN:=power@row1, IN:=TempDINTPrint:VD236, ENO=>power, OUT=>TempIntPrint:VW60]  c6 --  c7 [ EN:=power@row1, IN:=TempIntPrint:VW60, ENO=>?0_20_0, OUT=>VW412]
// row 2: c1 [box]  c3 [box]  c5 [box]  c7 [box]
// row 3: c1 [box]  c3 [box]  c7 [box]
// row 4: c3 [box]
Network 10
// (network saved uncompiled; FBD cells follow)
// row 0: c1 [MUL_R ]  c4 [ROUND ]  c7 [DI_I ]  c10 [MOV_W ]
// row 1: c1 [ EN:=Always_On:SM0.0, IN1:=PressureFinalVal:VD124, IN2:=10.0, ENO=>power, OUT=>PressRealPrint:VD240]  c2 --  c3 --  c4 [ EN:=power@row1, IN:=PressRealPrint:VD240, ENO=>power, OUT=>PressDINTPrint:VD244]  c5 --  c6 --  c7 [ EN:=power@row1, IN:=PressDINTPrint:VD244, ENO=>power, OUT=>PressIntPrint:VW62]  c8 --  c9 --  c10 [ EN:=power@row1, IN:=PressIntPrint:VW62, ENO=>V?0, OUT=>VW414]
// row 2: c1 [box]  c4 [box]  c7 [box]  c10 [box]
// row 3: c1 [box]
Network 11
// (network saved uncompiled; FBD cells follow)
// row 0: c1 [MOV_W ]
// row 1: c1 [ EN:=Always_On:SM0.0, IN:=SterTimePV:VW16, ENO=>?0_20_0, OUT=>VW416]
// row 2: c1 [box]
END_SUBROUTINE_BLOCK

DATA_BLOCK_TAB _PLC_DATA_1
BEGIN
VB1      16#2
VB3      16#1
VB5      16#3
VB7      16#1
VB25     16#8
VB27     16#5
VB33     16#3
VB102    16#19
VB103    16#6B
VB104    16#42
VB105    16#82
VB106    16#23
VB107    16#D7
VB108    16#42
VB109    16#80
VB112    16#42
VB113    16#9A
VB116    16#C3
VB117    16#D7
VB124    16#C3
VB125    16#C5
VB126    16#68
VB130    16#2F
VB131    16#87
VB132    16#42
VB133    16#F3
VB134    16#57
VB135    16#A
VB140    16#43
VB141    16#8A
VB142    16#33
VB148    16#42
VB149    16#C8
VB152    16#42
VB153    16#30
VB154    16#1B
VB155    16#6B
VB156    16#C3
VB157    16#AF
VB160    16#42
VB161    16#34
VB164    16#C3
VB165    16#C8
VB168    16#42
VB169    16#48
VB204    16#45
VB205    16#CB
VB206    16#58
VB208    16#46
VB209    16#3E
VB210    16#1C
END_DATA_BLOCK_TAB

DATA_BLOCK_TAB _PLC_DATA_2
BEGIN
VB21     16#1
VB23     16#9
VB143    16#33
VB188    16#40
VB189    16#2C
VB190    16#BC
VB191    16#30
VB192    16#3F
VB193    16#AC
VB194    16#BC
VB195    16#30
VB199    16#1
VB200    16#42
VB201    16#36
VB212    16#42
VB213    16#30
VB214    16#14
VB215    16#1
VB216    16#C3
VB217    16#C5
VB218    16#92
END_DATA_BLOCK_TAB

DATA_BLOCK_TAB _PLC_DATA_3
BEGIN
VB219    16#70
END_DATA_BLOCK_TAB

DATA_BLOCK_TAB _PLC_DATA_4
BEGIN
VB37     16#1
VB41     16#0
VB127    16#B8
END_DATA_BLOCK_TAB

DATA_BLOCK_TAB _PLC_DATA_5
BEGIN
VB9      16#2
VB11     16#1
VB43     16#5
VB172    16#C3
VB173    16#AF
VB176    16#42
VB177    16#34
VB180    16#C3
VB181    16#C8
VB220    16#40
VB221    16#A0
END_DATA_BLOCK_TAB

DATA_BLOCK_TAB _PLC_DATA_6
BEGIN
VB45     16#0
VB47     16#33
VB224    16#C3
VB225    16#C5
END_DATA_BLOCK_TAB

DATA_BLOCK_TAB _PLC_DATA_7
BEGIN
VB114    16#66
VB115    16#66
END_DATA_BLOCK_TAB

DATA_BLOCK_TAB _PLC_DATA_8
BEGIN
VB13     16#6
VB15     16#2
VB49     16#7
VB51     16#5
VB53     16#2
VB55     16#1
VB57     16#1
VB59     16#1
VB184    16#42
VB185    16#48
VB228    16#C3
VB229    16#C8
END_DATA_BLOCK_TAB

DATA_BLOCK_TAB _PLC_DATA_9
BEGIN
VB39     16#0
END_DATA_BLOCK_TAB

// (further data pages could not be read)
